FUNCTION_BLOCK IA_PosDeltaHighPrecRapidUpd (* ISOBUS Adapter for Position Delta, High Precision Rapid Update *)
  (* Standard: NMEA 2000; Classification: PGN 129027; Description: Copyright (c) 2024-2026 HR Agrartechnik GmbH This program and the accompanying materials are made available under the terms of the Eclipse Public License 2.0 which is available at https://www.eclipse.org/legal/epl-2.0/ SPDX-License-Identifier: EPL-2.0 *)
  (* Version 1.1, 2026-09-17, Franz Höpfinger, HR Agrartechnik GmbH, Bugfix (Franz: 'IA_VDS hat einen Bug, moeglicherweise alle anderen auch'): .IND->TIMEOUT.E1 ergaenzt (analog IA_VDS) - bisher wurde TIMEOUT.E1 NUR von .TIMEOUT gefeuert (Timeout-Beginn), nie beim Eintreffen einer normalen Botschaft (.IND) - TIMEOUT.D1 (Q_timeout=FALSE) wurde also gesetzt, aber nie an den TIMEOUT-Plug propagiert, sobald der Timeout wieder endete. *)
  (* Version 1.0, 2026-04-19, Franz Höpfinger, HR Agrartechnik GmbH, initial API and implementation (Adapter Wrapper for I_PosDeltaHighPrecRapidUpd) *)
  PACKAGE isobus::tecu;
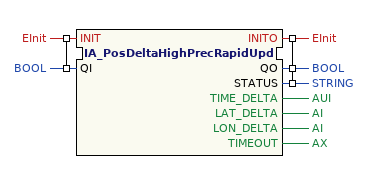
  EVENT_INPUT
    INIT : EInit WITH QI; (* Service Initialization *)
  END_EVENT
  EVENT_OUTPUT
    INITO : EInit WITH QO, STATUS; (* Initialization Confirm *)
  END_EVENT
  VAR_INPUT
    QI : BOOL; (* Event Input Qualifier *)
  END_VAR
  VAR_OUTPUT
    QO : BOOL; (* Event Output Qualifier *)
    STATUS : STRING;
  END_VAR
  PLUGS
    TIME_DELTA : adapter::types::unidirectional::AUI; (* Time Delta *)
    LAT_DELTA : adapter::types::unidirectional::AI; (* Latitude Delta *)
    LON_DELTA : adapter::types::unidirectional::AI; (* Longitude Delta *)
    TIMEOUT : adapter::types::unidirectional::AX; (* Timeout Status *)
  END_PLUGS
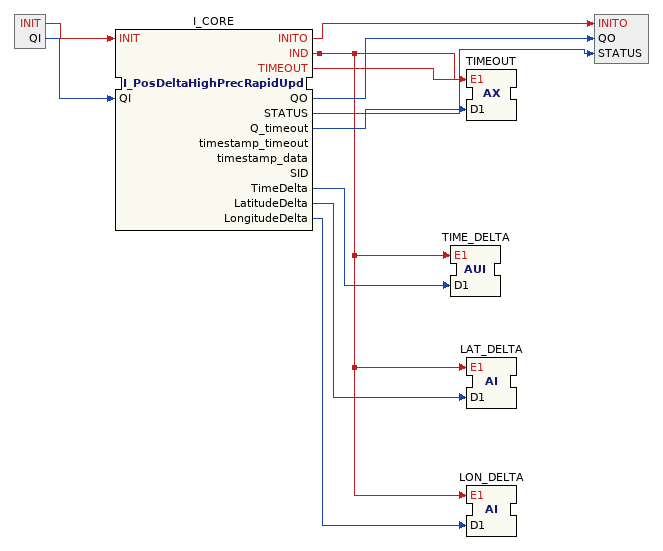
  FBS
    I_CORE : isobus::tecu::I_PosDeltaHighPrecRapidUpd;
  END_FBS
  EVENT_CONNECTIONS
    INIT TO I_CORE.INIT;
    I_CORE.INITO TO INITO;
    I_CORE.IND TO TIME_DELTA.E1;
    I_CORE.IND TO LAT_DELTA.E1;
    I_CORE.IND TO LON_DELTA.E1;
    I_CORE.TIMEOUT TO TIMEOUT.E1;
    I_CORE.IND TO TIMEOUT.E1;
  END_CONNECTIONS
  DATA_CONNECTIONS
    QI TO I_CORE.QI;
    I_CORE.QO TO QO;
    I_CORE.STATUS TO STATUS;
    I_CORE.TimeDelta TO TIME_DELTA.D1;
    I_CORE.LatitudeDelta TO LAT_DELTA.D1;
    I_CORE.LongitudeDelta TO LON_DELTA.D1;
    I_CORE.Q_timeout TO TIMEOUT.D1;
  END_CONNECTIONS
END_FUNCTION_BLOCK
